TYPE DUT_MODULE_INTERFACE_INPUT :
STRUCT
	///Mode to run (init,auto,manual,..)
	Mode: DUT_MODE;
	///check if the modules is alive
	ConnectionTestInput: BOOL;
	///Modules get their position
	PositionInput: LREAL;
	///Update data= TRUE, No updatedata=FALSE
	Watchbit: BOOL;
	///Emergency stop
	EmergencyStop: BOOL;
	///Range of INPUT skills
	SkillInput: ARRAY[0..SkillCnt] OF DUT_SKILL_INPUT;
END_STRUCT
END_TYPE

(* stored: Version 1.1.0.1, ProductVersion 3.1.0.25
   DUT DUT_MODULE_INTERFACE_INPUT: Id {d15d6b59-dbc2-4b17-a8b6-79dcb947d26b} *)
